{attribute 'qualified_only'}
{attribute 'strict'}
{attribute 'to_string'}
TYPE EWaferSize :
(
	Unknown := 0,
	_50mm := 50,
	_100mm := 100,
	_150mm := 150,
	_200mm := 200,
	_300mm := 300
);
END_TYPE

(* stored: Version 1.1.0.1, ProductVersion 3.1.4024.12
   DUT EWaferSize: Id {10b5bedd-7be1-4d77-af65-4c8e3bffe093} *)
